(* PLC project CoDeSys External Library Template, WAGO e!COCKPIT e!COCKPIT, author 3S - Smart Software Solutions GmbH *)
(* stored: creationDateTime 2019-10-29T12:22:40.5849973, version 3.5.5.30, modificationDateTime 2019-10-24T14:40:07.960949, organization 3S - Smart Software Solutions GmbH *)
(* Library project template with all possible element types, docu and a sample project structure *)

TYPE typModbusOdczytZapisZadanie : STRUCT
  bAdresUrzadzenia : BYTE;  (* ID urządzenia SLAVE w sieci MODBUS *)
  bFunkcja : BYTE;  (* kod funkcji użytej w rozkazie MODBUS *)
  uiAdresRejestru : UINT;  (* rejestr startowy *)
  pZmiennaDoOdczytu : POINTER TO WORD;  (* wskaźnik do zmiennej INT przechowującej wynik *)
  wWartoscDoZapisania : WORD;  (* wartość do zapisania *)
END_STRUCT;
END_TYPE
